% RSLogix 500 project P2_KOBIERSKI_M_v2.RSS, saved by version 8.30.00.16 %
PROJECT "UNTITLED"    % processor: Bul.1763 MicroLogix 1100 Series B %

PROGRAM FILES
  LAD 2 "MAIN"  4 rungs
  LAD 3 "IO"  8 rungs
  LAD 4 "CTRL"  7 rungs
  LAD 5 "CYCLE"  4 rungs

DATA FILES
  O0 OUTPUT  4 elements
  I1 INPUT  6 elements
  S2 STATUS  66 elements
  B3 BINARY  4 elements
  T4 TIMER  2 elements
  C5 COUNTER  1 elements
  R6 CONTROL  1 elements
  N7 INTEGER  1 elements
  F8 FLOAT  1 elements

LADDER 2 "MAIN"
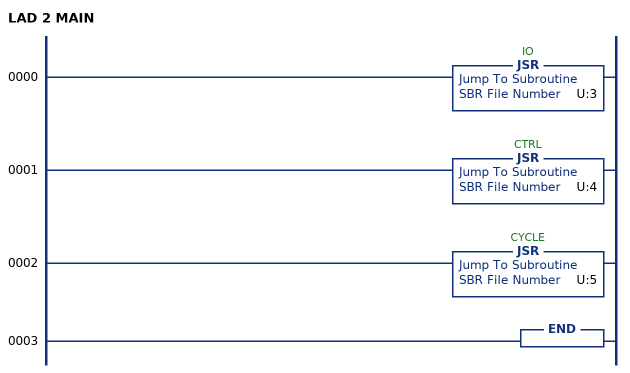
% Rung: 0 %
SOR JSR U:3 EOR
%   U:3  "IO" %
% Rung: 1 %
SOR JSR U:4 EOR
%   U:4  "CTRL" %
% Rung: 2 %
SOR JSR U:5 EOR
%   U:5  "CYCLE" %
% Rung: 3 %
SOR END EOR

LADDER 3 "IO"
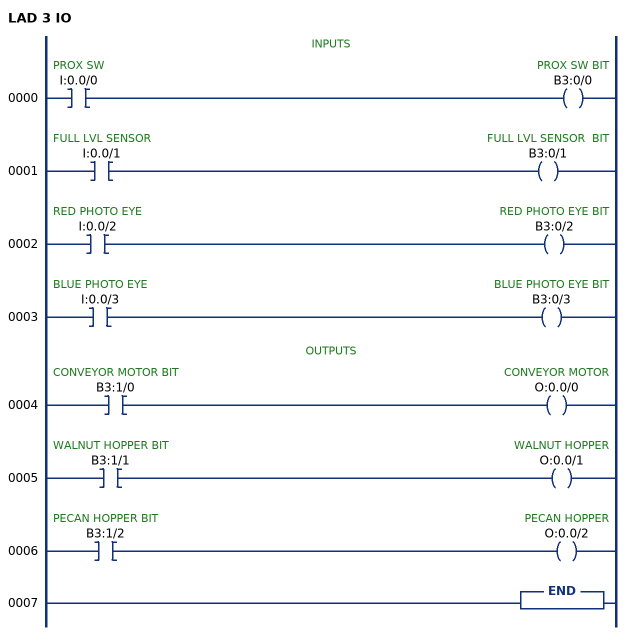
% Rung: 0 %
% INPUTS %
SOR XIC I:0.0/0 OTE B3:0/0 EOR
%   I:0.0/0  "PROX SW" %
%   B3:0/0  "PROX SW BIT" %
% Rung: 1 %
SOR XIC I:0.0/1 OTE B3:0/1 EOR
%   I:0.0/1  "FULL LVL SENSOR" %
%   B3:0/1  "FULL LVL SENSOR  BIT" %
% Rung: 2 %
SOR XIC I:0.0/2 OTE B3:0/2 EOR
%   I:0.0/2  "RED PHOTO EYE" %
%   B3:0/2  "RED PHOTO EYE BIT" %
% Rung: 3 %
SOR XIC I:0.0/3 OTE B3:0/3 EOR
%   I:0.0/3  "BLUE PHOTO EYE" %
%   B3:0/3  "BLUE PHOTO EYE BIT" %
% Rung: 4 %
% OUTPUTS %
SOR XIC B3:1/0 OTE O:0.0/0 EOR
%   B3:1/0  "CONVEYOR MOTOR BIT" %
%   O:0.0/0  "CONVEYOR MOTOR" %
% Rung: 5 %
SOR XIC B3:1/1 OTE O:0.0/1 EOR
%   B3:1/1  "WALNUT HOPPER BIT" %
%   O:0.0/1  "WALNUT HOPPER" %
% Rung: 6 %
SOR XIC B3:1/2 OTE O:0.0/2 EOR
%   B3:1/2  "PECAN HOPPER BIT" %
%   O:0.0/2  "PECAN HOPPER" %
% Rung: 7 %
SOR END EOR

LADDER 4 "CTRL"
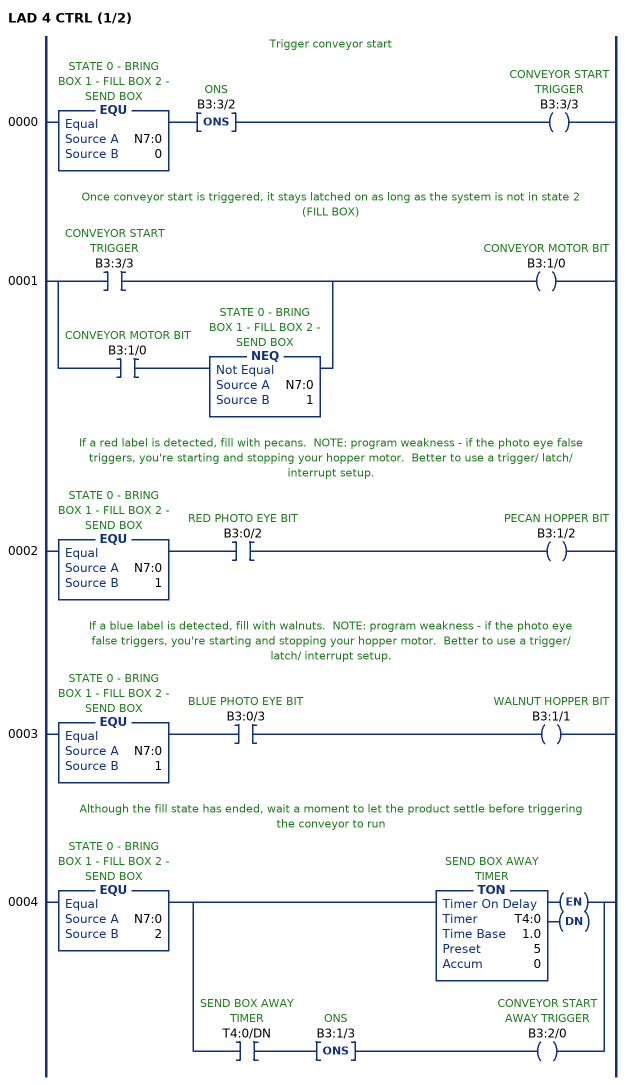
% Rung: 0 %
% Trigger conveyor start %
SOR EQU N7:0 0 ONS B3:3/2 OTE B3:3/3 EOR
%   N7:0  "STATE 0 - BRING BOX 1 - FILL BOX 2 - SEND BOX" %
%   B3:3/2  "ONS" %
%   B3:3/3  "CONVEYOR START TRIGGER" %
% Rung: 1 %
% Once conveyor start is triggered, it stays latched on as long as the system is not in state 2 (FILL BOX) %
SOR BST XIC B3:3/3 NXB XIC B3:1/0 NEQ N7:0 1 BND OTE B3:1/0 EOR
%   B3:3/3  "CONVEYOR START TRIGGER" %
%   B3:1/0  "CONVEYOR MOTOR BIT" %
%   N7:0  "STATE 0 - BRING BOX 1 - FILL BOX 2 - SEND BOX" %
% Rung: 2 %
% If a red label is detected, fill with pecans.  NOTE: program weakness - if the photo eye false triggers, you're starting and stopping your hopper motor.  Better to use a trigger/ latch/ interrupt setup. %
SOR EQU N7:0 1 XIC B3:0/2 OTE B3:1/2 EOR
%   N7:0  "STATE 0 - BRING BOX 1 - FILL BOX 2 - SEND BOX" %
%   B3:0/2  "RED PHOTO EYE BIT" %
%   B3:1/2  "PECAN HOPPER BIT" %
% Rung: 3 %
% If a blue label is detected, fill with walnuts.  NOTE: program weakness - if the photo eye false triggers, you're starting and stopping your hopper motor.  Better to use a trigger/ latch/ interrupt setup. %
SOR EQU N7:0 1 XIC B3:0/3 OTE B3:1/1 EOR
%   N7:0  "STATE 0 - BRING BOX 1 - FILL BOX 2 - SEND BOX" %
%   B3:0/3  "BLUE PHOTO EYE BIT" %
%   B3:1/1  "WALNUT HOPPER BIT" %
% Rung: 4 %
% Although the fill state has ended, wait a moment to let the product settle before triggering the conveyor to run %
SOR EQU N7:0 2 BST TON T4:0 1.0 5 0 NXB XIC T4:0/DN ONS B3:1/3 OTE B3:2/0 BND EOR
%   N7:0  "STATE 0 - BRING BOX 1 - FILL BOX 2 - SEND BOX" %
%   T4:0  "SEND BOX AWAY TIMER" %
%   B3:1/3  "ONS" %
%   B3:2/0  "CONVEYOR START AWAY TRIGGER" %

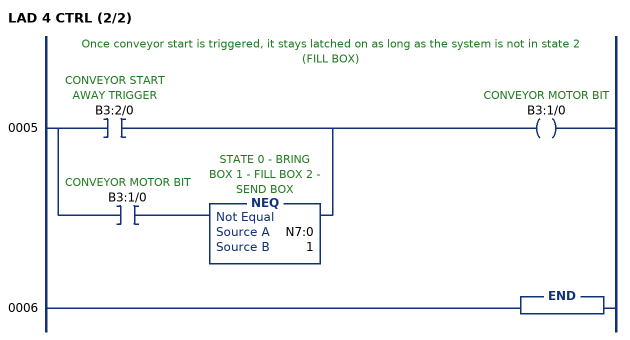
% Rung: 5 %
% Once conveyor start is triggered, it stays latched on as long as the system is not in state 2 (FILL BOX) %
SOR BST XIC B3:2/0 NXB XIC B3:1/0 NEQ N7:0 1 BND OTE B3:1/0 EOR
%   B3:2/0  "CONVEYOR START AWAY TRIGGER" %
%   B3:1/0  "CONVEYOR MOTOR BIT" %
%   N7:0  "STATE 0 - BRING BOX 1 - FILL BOX 2 - SEND BOX" %
% Rung: 6 %
SOR END EOR

LADDER 5 "CYCLE"
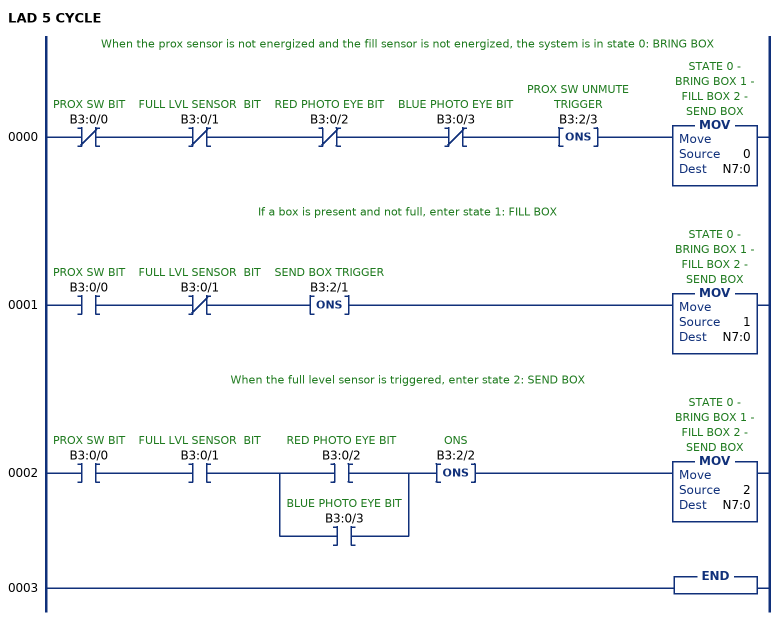
% Rung: 0 %
% When the prox sensor is not energized and the fill sensor is not energized, the system is in state 0: BRING BOX %
SOR XIO B3:0/0 XIO B3:0/1 XIO B3:0/2 XIO B3:0/3 ONS B3:2/3 MOV 0 N7:0 EOR
%   B3:0/0  "PROX SW BIT" %
%   B3:0/1  "FULL LVL SENSOR  BIT" %
%   B3:0/2  "RED PHOTO EYE BIT" %
%   B3:0/3  "BLUE PHOTO EYE BIT" %
%   B3:2/3  "PROX SW UNMUTE TRIGGER" %
%   N7:0  "STATE 0 - BRING BOX 1 - FILL BOX 2 - SEND BOX" %
% Rung: 1 %
% If a box is present and not full, enter state 1: FILL BOX %
SOR XIC B3:0/0 XIO B3:0/1 ONS B3:2/1 MOV 1 N7:0 EOR
%   B3:0/0  "PROX SW BIT" %
%   B3:0/1  "FULL LVL SENSOR  BIT" %
%   B3:2/1  "SEND BOX TRIGGER" %
%   N7:0  "STATE 0 - BRING BOX 1 - FILL BOX 2 - SEND BOX" %
% Rung: 2 %
% When the full level sensor is triggered, enter state 2: SEND BOX %
SOR XIC B3:0/0 XIC B3:0/1 BST XIC B3:0/2 NXB XIC B3:0/3 BND ONS B3:2/2 MOV 2 N7:0 EOR
%   B3:0/0  "PROX SW BIT" %
%   B3:0/1  "FULL LVL SENSOR  BIT" %
%   B3:0/2  "RED PHOTO EYE BIT" %
%   B3:0/3  "BLUE PHOTO EYE BIT" %
%   B3:2/2  "ONS" %
%   N7:0  "STATE 0 - BRING BOX 1 - FILL BOX 2 - SEND BOX" %
% Rung: 3 %
SOR END EOR

OTHER DOCUMENTED ADDRESSES
  B3:1/4  "SEND BOX AWAY TRIGGER"
  B3:1/5  "ONS"
  B3:2/4  "MUTE PROX SW"
  B3:3/4  "ONS"
  B3:3/5  "FILL START TRIGGER"
  N7:0/1  "STATE 0 - BRING BOX 1 - FILL BOX 2 - SEND BOX"
  T4:1  "PROX SW MUTE TIMER"

COMMENTS NOT ATTACHED TO A CURRENT RUNG
  B3:1/2: If a box is present and not full, and the label is red, fill with pecans.
  B3:1/1: If a box is present and not full, and the label is blue, fill with walnuts.
  B3:1/0: Conveyor Run command: When the PROX SW and the LVL SENSOR are off, run the conveyor. On BOX FULL, run the conveyor until the PROX SW is triggered (outside of MUTED period).
  B3:2/1: Once a box is full, delay a moment to catch and final falling product then trigger the BOX FULL signal.
  T4:1: When PROX SW and FULL LVL SENSOR are both on, 1) short delay to catch final falling product; 2) longer delay muting the PROX SW bit to let the box pass.
  B3:3/0: When the prox sensor is energized, and the box is not full, fill the box.

DATA TABLE (non-zero values as saved)
DATA T4
% .PRE .ACC %
% T4:0 % 5 0
% T4:1 % 5 0
